// TIA Portal V20 export
DATA_BLOCK "PNDevDiagInterface_X1"   // DB261
// stored: InstanceOfName LAF_typeDevDiagInterface, InstanceOfType UDT
"LAF_typeDevDiagInterface"
   // VAR
   //    globalInfoHmi : "LAF_typeDevDiagGlobal";
   //    devStateHmi { ExternalWritable := 'False'} : Array[0..256] of "LAF_typeDevDiagBasic";
   //    devStateUser { ExternalAccessible := 'False'; ExternalVisible := 'False'; ExternalWritable := 'False'} : Array[0..256] of "LAF_typeDevDiagState";
   // END_VAR
BEGIN
   globalInfoHmi.geoAddressSystem := 0;
   globalInfoHmi.maxDevices := 0;
   globalInfoHmi.maxModuls := 0;
   globalInfoHmi.lowestDevNoConfig := 0;
   globalInfoHmi.highestDevNoConfig := 0;
   globalInfoHmi.numberOfDevices.configured := 0;
   globalInfoHmi.numberOfDevices.notPresent := 0;
   globalInfoHmi.numberOfDevices.deactivated := 0;
   globalInfoHmi.numberOfDevices.faulty := 0;
   globalInfoHmi.numberOfDevices.problem := 0;
   globalInfoHmi.devDiagSummary := FALSE;
   globalInfoHmi.blockBusyAfterNewStart := FALSE;
   globalInfoHmi.manualReadAll := FALSE;
   globalInfoHmi.resetHistoryAll := FALSE;
   devStateHmi[0..256].devNumber := 0;
   devStateHmi[0..256].devName := '';
   devStateHmi[0..256].devStateDezCoded := 0;
   devStateHmi[0..256].devStateBitCoded := 16#0000;
   devStateHmi[0..256].first8CharOfMlfb := '';
   devStateUser[0..256].configured := FALSE;
   devStateUser[0..256].faulty := FALSE;
   devStateUser[0..256].deactivated := FALSE;
   devStateUser[0..256].present := FALSE;
   devStateUser[0..256].problem := FALSE;
   devStateUser[0..256].networkError := FALSE;
   devStateUser[0..256].maintenanceRequired := FALSE;
   devStateUser[0..256].maintenanceDemanded := FALSE;
   devStateUser[0..256].wasFaulty := FALSE;
   devStateUser[0..256].wasProblem := FALSE;
   devStateUser[0..256].modulStateSummary := FALSE;
   devStateUser[0..256].spare11 := FALSE;
   devStateUser[0..256].spare12 := FALSE;
   devStateUser[0..256].spare13 := FALSE;
   devStateUser[0..256].spare14 := FALSE;
   devStateUser[0..256].spare15 := FALSE;
END_DATA_BLOCK
